			// code that is repeated every cycle in this state
				iCharacteristicAt2				:= aTransferPackages[0].iTransferValue;
				iCharacteristicAt4				:= aTransferPackages[1].iTransferValue;
				iOptProportionalGainFor2		:= aTransferPackages[2].iTransferValue;
				iOptIntegralGainFor2			:= aTransferPackages[3].iTransferValue;
				iOptTimeConstantFor2			:= aTransferPackages[4].iTransferValue;
				iOptShiftZeroPointSwitchOff2	:= aTransferPackages[5].iTransferValue;
				iOptProportionalGainFor4		:= aTransferPackages[6].iTransferValue;
				iOptIntegralGainFor4			:= aTransferPackages[7].iTransferValue;
				iOptTimeConstantFor4			:= aTransferPackages[8].iTransferValue;
				iOptShiftZeroPointSwitchOff4	:= aTransferPackages[9].iTransferValue;
				iInPortRetracted_optional		:= aTransferPackages[10].iTransferValue;
				iInPortAdvanced_optional		:= aTransferPackages[11].iTransferValue;
			//-----------------------------------------------------------------------------------------------------------
			
			// Transition
				xStateChange := TRUE;
				iState := 50;
				iCommandNumber := 40;
			//-----------------------------------------------------------------------------------------------------------
		
		50:	// DONE
			// code that is executed only in the first cycle of this state
				IF xStateChange = TRUE THEN
					xStateChange := FALSE;
					iResponse := eTransferResponse.transfer_successful;
					xDone := TRUE;
					xError := FALSE;
					xBusy := FALSE;
					xAborted := FALSE;
				END_IF
			//-----------------------------------------------------------------------------------------------------------
			
			// code that is repeated every cycle in this state	
				IF fbuploadMultipleParameters.xExecute = FALSE  AND fbuploadMultipleParameters.xUploadDone = FALSE AND fbuploadMultipleParameters.xUploadError = FALSE AND iCurrentValveMode = 63 THEN		//FB_UploadMultipleParameters was reset
					iCommandNumber := 5;	// exit transfer mode
				END_IF
			//-----------------------------------------------------------------------------------------------------------
			
			// Transition
				IF fbuploadMultipleParameters.xExecute = FALSE  AND fbuploadMultipleParameters.xUploadDone = FALSE AND fbuploadMultipleParameters.xUploadError = FALSE AND xExecute = FALSE THEN
					xStateChange := TRUE;
					iState := 100;
				END_IF
			//-----------------------------------------------------------------------------------------------------------
			
		70:	// ERROR
			// code that is executed only in the first cycle of this state
				IF xStateChange = TRUE THEN
					xStateChange := FALSE;
					//iResponse := eTransferResponse.communication_failed;	// set within the transition of the last state
					xDone := FALSE;
					xError := TRUE;
					xBusy := FALSE;
					xAborted := FALSE;
				END_IF
			//-----------------------------------------------------------------------------------------------------------
			
			// code that is repeated every cycle in this state	
			//-----------------------------------------------------------------------------------------------------------
			
			// Transition
				IF xExecute = FALSE AND xAbort = FALSE THEN
					xStateChange := TRUE;
					iState := 100;
				END_IF
			//-----------------------------------------------------------------------------------------------------------
			
		80:	// ABORTING
			// code that is executed only in the first cycle of this state
				IF xStateChange = TRUE THEN
					xStateChange := FALSE;
					iResponse := eTransferResponse.aborting;
					xBusy := FALSE;
					xDone := FALSE;
					xError := FALSE;
					xAborted := TRUE;
				END_IF
			//-----------------------------------------------------------------------------------------------------------
			
			// code that is repeated every cycle in this state
				IF iCurrentValveMode = 63 THEN
					iCommandNumber := 5;	// exit transfer mode
				ELSIF iCurrentValveMode <> 61 AND iCurrentValveMode <> 63 THEN
					iCommandNumber := 6;	// stop running motion apps
				ELSE
					iCommandNumber := 0; 
				END_IF
			//-----------------------------------------------------------------------------------------------------------
			
			// Transition
				IF xAbort = FALSE AND xExecute = FALSE AND iCurrentValveMode = 61 THEN
					xStateChange := TRUE;
					iState := 100;
				END_IF
			//-----------------------------------------------------------------------------------------------------------

		100:	// RESETTING FUNCTION BLOCK AND VALVE
			// code that is executed only in the first cycle of this state
				IF xStateChange = TRUE THEN
					xStateChange := FALSE;
					iResponse := eTransferResponse.resetting;
					xDone := FALSE;
					xError := FALSE;
					xBusy := FALSE;
					xAborted := FALSE;
				END_IF
			//-----------------------------------------------------------------------------------------------------------
			
			// code that is repeated every cycle in this state	
				IF iCurrentValveMode = 63 THEN
					iCommandNumber := 5;	// exit transfer mode
				ELSIF iCurrentValveMode <> 61 AND iCurrentValveMode <> 63 THEN
					iCommandNumber := 6;	// stop running motion apps
				END_IF
				
				// reset funktion block fbreadmultipleparameters
				// not done via command number because this is used to reset valve
					fbuploadMultipleParameters(
						awBusDataFromVTEM:= awBusDataFromVTEM, 
						awBusDataToVTEM:= awBusDataToVTEM, 
						xExecute:= FALSE, 
						iResponse=> , 
						iCurrentValue=> , 
						xUploadDone=> , 
						xUploadError=> , 
						aTransferPackages:= aTransferPackages);
				
				// reset parameter outputs
					iParameterSet := 1;
					iCharacteristicAt2 := 0;
					iCharacteristicAt4 := 0;
					iOptProportionalGainFor2 := 0;
					iOptIntegralGainFor2 := 0;
					iOptTimeConstantFor2 := 0;
					iOptShiftZeroPointSwitchOff2 := 0;
					iOptProportionalGainFor4 := 0;
					iOptIntegralGainFor4 := 0;
					iOptTimeConstantFor4 := 0;
					iOptShiftZeroPointSwitchOff4 := 0;
					iInPortRetracted_optional := 0;
					iInPortAdvanced_optional := 0;
				
				// reset parameter array
					FOR iCounterResetArray := 0 TO 100 BY 1 DO
						aTransferPackages[iCounterResetArray].iChannel := 0;
						aTransferPackages[iCounterResetArray].iAddressedTarget := 0;
						aTransferPackages[iCounterResetArray].iIndex := 0;
						aTransferPackages[iCounterResetArray].iTransferValue := 0;
					END_FOR
					
					iCounterResetArray := 0;
					xFirstCycle := TRUE;
			//-----------------------------------------------------------------------------------------------------------
			
			// Transition
				IF iCurrentValveMode = 61 THEN
					iCommandNumber := 6; // Last command to send before the FB is in IDLE
					xStateChange := TRUE;
					iState := 10;
				END_IF
			//-----------------------------------------------------------------------------------------------------------
			
	END_CASE
//-----------------------------------------------------------------------------------------------------------

// Command section
	CASE iCommandNumber OF
		0:	// IDLE
			;
		
		5:	// EXIT TRANSFER MODE
			fbwritevaluetoword(iValue:=63, iStartBit:=0, iEndBit:=5, wDataWord:=awBusDataToVTEM[0], xError=> );							// Valve Mode = 63
			fbwritevaluetoword(iValue:=0, iStartBit:=6, iEndBit:=7, wDataWord:=awBusDataToVTEM[0], xError=> );							// 0 (unused)
			fbwritevaluetoword(iValue:=0, iStartBit:=8, iEndBit:=12, wDataWord:=awBusDataToVTEM[0], xError=> );							// Channel = 0 (ignored)
			fbwritevaluetoword(iValue:=3, iStartBit:=13, iEndBit:=15, wDataWord:=awBusDataToVTEM[0], xError=> );						// Transfer Control = 3 (Exit transfer mode)
			fbwritevaluetoword(iValue:=0, iStartBit:=0, iEndBit:=7, wDataWord:=awBusDataToVTEM[1], xError=> );							// Addressed Target = 0 (ignored)
			fbwritevaluetoword(iValue:=0, iStartBit:=8, iEndBit:=15, wDataWord:=awBusDataToVTEM[1], xError=> );							// Index = 0 (ignored)
			fbwritevaluetoword(iValue:=0, iStartBit:=0, iEndBit:=15, wDataWord:=awBusDataToVTEM[2], xError=> );							// Value = 0 (ignored)
			
		6:	// STOP RUNNING MOTION APP
			fbwritevaluetoword(iValue:=61, iStartBit:=0, iEndBit:=5, wDataWord:=awBusDataToVTEM[0], xError=> );							// Valve Mode = 61 (stop)
			fbwritevaluetoword(iValue:=0, iStartBit:=6, iEndBit:=7, wDataWord:=awBusDataToVTEM[0], xError=> );							// App Control = 0 (unused)
			fbwritevaluetoword(iValue:=0, iStartBit:=8, iEndBit:=15, wDataWord:=awBusDataToVTEM[0], xError=> );							// App Option = 0 (unused)
			fbwritevaluetoword(iValue:=0, iStartBit:=0, iEndBit:=15, wDataWord:=awBusDataToVTEM[1], xError=> );							// Setpoint Value 1 = 0 (unused)
			fbwritevaluetoword(iValue:=0, iStartBit:=0, iEndBit:=15, wDataWord:=awBusDataToVTEM[2], xError=> );							// Setpoint Value 2 = 0 (unused)
		
		30:	// RUN FB_UPLOADMULTIPLEPARAMETERS
			fbuploadMultipleParameters(
				awBusDataFromVTEM:= awBusDataFromVTEM, 
				awBusDataToVTEM:= awBusDataToVTEM, 
				xExecute:= TRUE, 
				iResponse=> , 
				iCurrentValue=> , 
				xUploadDone=> , 
				xUploadError=> , 
				aTransferPackages:= aTransferPackages);

		40:	// RESET FB_UPLOADMULTIPLEPARAMETERS
			fbuploadMultipleParameters(
				awBusDataFromVTEM:= awBusDataFromVTEM, 
				awBusDataToVTEM:= awBusDataToVTEM, 
				xExecute:= FALSE, 
				iResponse=> , 
				iCurrentValue=> , 
				xUploadDone=> , 
				xUploadError=> , 
				aTransferPackages:= aTransferPackages);
	END_CASE
//-----------------------------------------------------------------------------------------------------------

END_FUNCTION_BLOCK

// Transfermode/specific_MA_config/FB_Read_config_MA_04
/// This function block can be used to upload the configuration of Motion App 4 ("Model-based proportional pressure regulation").
/// The specific parameters of this Motion App are the outputs of this FB
/// The function block uses the transfer mode to read this configuration from the Motion Terminal
/// and indicates the state of the upload process at the output iResponse.

FUNCTION_BLOCK FB_Read_config_MA_04
VAR_INPUT
	awBusDataFromVTEM 				: ARRAY [0..2] OF WORD;		// array of 3 words of process data received from the Motion Terminal
END_VAR
	
VAR_IN_OUT
	awBusDataToVTEM 				: ARRAY [0..2] OF WORD; 	// array of 3 words of process data sent to the Motion Terminal
END_VAR

VAR_INPUT
	xExecute 						: BOOL; 					// rising edge starts the reading process, falling edge resets the function block after reading is done
	xAbort							: BOOL;						// rising edge aborts the reading process
	iParameterSet					: INT := 1; 				// the parameter set to be read from, 1 by default
END_VAR                     		

VAR_OUTPUT                  		
	// system parameters
		iTubingLengthAt2 			: INT; 						// length of the tubing connected to outlet port 2 of the valve [1 digit = 1 mm]
		iTubingLengthAt4 			: INT;						// length of the tubing connected to outlet port 4 of the valve [1 digit = 1 mm]
		iTubingInnerDiameterAt2 	: INT;  					// inner diameter of the tubing connected to outlet port 2 of the valve [1 digit = 0.01 mm]
		iTubingInnerDiameterAt4 	: INT;						// inner diameter of the tubing connected to outlet port 4 of the valve [1 digit = 0.01 mm]
		iVolumeAt2 					: INT; 						// size/capacity of the volume connected to outlet port 2 of the valve [1 digit = 0.001 l]
	 	iVolumeAt4 					: INT;						// size/capacity of the volume connected to outlet port 4 of the valve [1 digit = 0.001 l]
		iInPortRetracted_optional	: INT;						// Sensor port for detection of end position at pressurisation of outlet port 2 (retracted), value is number of the slot (beginning from 0 and including valve slots) * 10 + number of the port
		iInPortAdvanced_optional	: INT;						// Sensor port for detection of end position at pressurisation of outlet port 4 (advanced), value is number of the slot (beginning from 0 and including valve slots) * 10 + number of the port
		
	// application parameters
		iPressureRiseAt2 			: INT; 						// maximum pressure rise at outlet port 2 [1 digit = 0.01 bar/s]
		iPressureRiseAt4 			: INT;						// maximum pressure rise at outlet port 4 [1 digit = 0.01 bar/s]
		
	// function block response
		iResponse 					: eTransferResponse; 		// returns the status of the upload process
		xBusy						: BOOL;						// TRUE as long as the upload process is running
		xDone 						: BOOL; 					// indicates whether the upload was successfull
		xError 						: BOOL; 					// indicates whether an error occurred during the transfer
		xAborted					: BOOL;						// TRUE if the function block was canceled by xAbort	
END_VAR

VAR
	iState							: INT := 10;
	xStateChange					: BOOL;
	iCommandNumber					: INT;
	xFirstCycle						: BOOL := TRUE;				// indicator for the first cycle of the function block
	iParameterSetFC					: INT;						// value on input iParameterSet during first cycle
	
	aTransferPackages				: ARRAY [0..100] OF stTransferPackage;
	fbreadbitsfromword				: FB_Read_Bits_From_Word;
	fbuploadMultipleParameters 		: FB_Upload_Multiple_Parameters;
	fbWriteValueToWord 				: FB_Write_Value_To_Word;

	iCounterResetArray				: INT;

	iCurrentValveMode				: INT;						//
END_VAR

(*****************************************************************************************************

Festo SE & Co. KG, Esslingen
Copyright (c) 2021. All rights reserved.

Product:            Motion Terminal VTEM
Description:        Function Block to upload the parameters for Motion App 4 from the Motion Terminal

Object version:     2.00
Last change:        2021-07
======================================================================================================
                                       H I S T O R Y
======================================================================================================
Version:            2.00
Date:               2021-07
Change/Activity:    - created (#3872357)
Release:            3.5.7.237 (CODESYS 3.5.7.2, Lib version 3.7)
Author:             JEBU
======================================================================================================

*****************************************************************************************************)

// pre-check of the value for the parameter set
	IF xExecute = TRUE AND (iParameterSet < 1 OR iParameterSet > 5) THEN		// invalid input for the parameter set
		xDone := FALSE; 
		xError := TRUE; 
		iResponse := eTransferResponse.invalid_ParameterSet;
		xStateChange := TRUE;
		iState := 70;	// ERROR
	END_IF
//-----------------------------------------------------------------------------------------------------------

// check if iParameterSet was changed
	IF xExecute = TRUE AND xFirstCycle = TRUE THEN
		xFirstCycle := FALSE;
		iParameterSetFC := iParameterSet;
	END_IF
	
	IF xExecute = TRUE AND iParameterSet <> iParameterSetFC THEN
		xStateChange := TRUE;
		iState := 70;
		iResponse := eTransferResponse.FB_needs_rising_edge_xExecute;
	END_IF
//-----------------------------------------------------------------------------------------------------------

// WRITE PARAMETER INDICES INTO ARRAY
	//iTubingLengthAt2
		aTransferPackages[0].iChannel := iParameterSet;
		aTransferPackages[0].iAddressedTarget := 4;
		aTransferPackages[0].iIndex := 12;
	
	//iTubingLengthAt4
		aTransferPackages[1].iChannel := iParameterSet;
		aTransferPackages[1].iAddressedTarget := 4;
		aTransferPackages[1].iIndex := 13;
	
	//iTubingInnerDiameterAt2
		aTransferPackages[2].iChannel := iParameterSet;
		aTransferPackages[2].iAddressedTarget := 4;
		aTransferPackages[2].iIndex := 14;
	
	//iTubingInnerDiameterAt4
		aTransferPackages[3].iChannel := iParameterSet;
		aTransferPackages[3].iAddressedTarget := 4;
		aTransferPackages[3].iIndex := 15;
	
	//iVolumeAt2
		aTransferPackages[4].iChannel := iParameterSet;
		aTransferPackages[4].iAddressedTarget := 4;
		aTransferPackages[4].iIndex := 40;
	
	//iVolumeAt4
		aTransferPackages[5].iChannel := iParameterSet;
		aTransferPackages[5].iAddressedTarget := 4;
		aTransferPackages[5].iIndex := 41;
	
	//iPressureRiseAt2
		aTransferPackages[6].iChannel := iParameterSet;
		aTransferPackages[6].iAddressedTarget := 4;
		aTransferPackages[6].iIndex := 182;
	
	//iPressureRiseAt4
		aTransferPackages[7].iChannel := iParameterSet;
		aTransferPackages[7].iAddressedTarget := 4;
		aTransferPackages[7].iIndex := 183;
	
	//iInPortRetract_optional
		aTransferPackages[8].iChannel := iParameterSet;
		aTransferPackages[8].iAddressedTarget := 4;
		aTransferPackages[8].iIndex := 70;
	
	//iInPortAdvanced_optional
		aTransferPackages[9].iChannel := iParameterSet;
		aTransferPackages[9].iAddressedTarget := 4;
		aTransferPackages[9].iIndex := 71;
	
	// define end of parameter list to be uploaded by setting all variables to 0 (end criterion for FB_Upload_Multiple_Parameters)
		aTransferPackages[10].iChannel := 0;
		aTransferPackages[10].iAddressedTarget := 0;
		aTransferPackages[10].iIndex := 0;
//-----------------------------------------------------------------------------------------------------------

// Read the current status of the the motion terminal
	fbreadbitsfromword(wData:= awBusDataFromVTEM[0], iStartBit:=0, iEndBit:= 5, iValue=> iCurrentValveMode, xError=> );				// read current valve mode
//-----------------------------------------------------------------------------------------------------------

// Transition: Aborting condition when xAbort is TRUE in all States except "IDLE" , "ABORTING" and "RESETTING"
	IF xAbort = TRUE AND NOT(iState = 10 AND xExecute = FALSE) AND iState <> 80 AND iState <> 100 THEN
		xStateChange := TRUE;	// Leaving current state
		iState := 80;	// Choosing next state, here: ABORTING
	END_IF
//-----------------------------------------------------------------------------------------------------------

// local state machine
	CASE iState OF
		10:	// IDLE
			// code that is executed only in the first cycle of this state
				IF xStateChange = TRUE THEN
					xStateChange := FALSE;
					iResponse := eTransferResponse.ready_for_new_transfer;
					xDone := FALSE;
					xError := FALSE;
					xBusy := FALSE;
					xAborted := FALSE;
				END_IF
			//-----------------------------------------------------------------------------------------------------------
			
			// code that is repeated every cycle in this state
				iCommandNumber := 0;
			//-----------------------------------------------------------------------------------------------------------
			
			// Transition
			IF xExecute = TRUE THEN
				xStateChange := TRUE;
				iState := 20;
			END_IF
			//-----------------------------------------------------------------------------------------------------------
		
		20:	// RESETTING VALVE MODE TO 61
			// code that is executed only in the first cycle of this state
				IF xStateChange = TRUE THEN
					xStateChange := FALSE;
					iResponse := eTransferResponse.preparing_transfer;
					xDone := FALSE;
					xError := FALSE;
					xBusy := TRUE;
					xAborted := FALSE;
				END_IF
			//-----------------------------------------------------------------------------------------------------------
			
			// code that is repeated every cycle in this state	
				IF iCurrentValveMode = 63 THEN
					iCommandNumber := 5;	// exit transfer mode
				ELSIF iCurrentValveMode <> 61 AND iCurrentValveMode <> 63 THEN
					iCommandNumber := 6;	// stop running motion apps
				END_IF 
			//-----------------------------------------------------------------------------------------------------------
			
			// Transition
				IF iCurrentValveMode = 61 THEN
					xStateChange := TRUE;	// Leave this state
					iState := 30;
					iCommandNumber := 30;			
				END_IF
			//-----------------------------------------------------------------------------------------------------------
		
		30:	// READING PARAMETER VALUES
			// code that is executed only in the first cycle of this state
				IF xStateChange = TRUE THEN
					xStateChange := FALSE;
					iResponse := eTransferResponse.transferring;
					xDone := FALSE;
					xError := FALSE;
					xBusy := TRUE;
					xAborted := FALSE;
				END_IF
			//-----------------------------------------------------------------------------------------------------------
			
			// code that is repeated every cycle in this state
				iCommandNumber := 30;		// read parameter values
			//-----------------------------------------------------------------------------------------------------------
			
			// Transition
				IF fbuploadMultipleParameters.xExecute = TRUE AND fbuploadMultipleParameters.xUploadDone = TRUE AND fbuploadMultipleParameters.xUploadError = FALSE THEN	// Upload Done
					xStateChange := TRUE;
					iState := 40;	// Write parameter values to outputs
				ELSIF fbuploadMultipleParameters.xExecute = TRUE AND fbuploadMultipleParameters.xUploadDone = FALSE AND fbuploadMultipleParameters.xUploadError = TRUE THEN	// Error during update
					xStateChange := TRUE;
					iState := 70;	// ERROR
					iResponse := fbuploadMultipleParameters.iResponse;
				END_IF
			//-----------------------------------------------------------------------------------------------------------
		
		40:	// WRITE PARAMETER VALUES TO OUTPUTS
			// code that is executed only in the first cycle of this state
				IF xStateChange = TRUE THEN
					xStateChange := FALSE;
					iResponse := eTransferResponse.transferring;
					xDone := FALSE;
					xError := FALSE;
					xBusy := TRUE;
					xAborted := FALSE;
				END_IF
			//-----------------------------------------------------------------------------------------------------------
			
			// code that is repeated every cycle in this state
				iTubingLengthAt2			:= aTransferPackages[0].iTransferValue;
				iTubingLengthAt4			:= aTransferPackages[1].iTransferValue;
				iTubingInnerDiameterAt2		:= aTransferPackages[2].iTransferValue;
				iTubingInnerDiameterAt4		:= aTransferPackages[3].iTransferValue;
				iVolumeAt2					:= aTransferPackages[4].iTransferValue;
				iVolumeAt4					:= aTransferPackages[5].iTransferValue;
				iPressureRiseAt2			:= aTransferPackages[6].iTransferValue;
				iPressureRiseAt4			:= aTransferPackages[7].iTransferValue;
				iInPortRetracted_optional	:= aTransferPackages[8].iTransferValue;
				iInPortAdvanced_optional	:= aTransferPackages[9].iTransferValue;
			//-----------------------------------------------------------------------------------------------------------
			
			// Transition
				xStateChange := TRUE;
				iState := 50;
				iCommandNumber := 40;
			//-----------------------------------------------------------------------------------------------------------
		
		50:	// DONE
			// code that is executed only in the first cycle of this state
				IF xStateChange = TRUE THEN
					xStateChange := FALSE;
					iResponse := eTransferResponse.transfer_successful;
					xDone := TRUE;
					xError := FALSE;
					xBusy := FALSE;
					xAborted := FALSE;
				END_IF
			//-----------------------------------------------------------------------------------------------------------
			
			// code that is repeated every cycle in this state	
				IF fbuploadMultipleParameters.xExecute = FALSE  AND fbuploadMultipleParameters.xUploadDone = FALSE AND fbuploadMultipleParameters.xUploadError = FALSE AND iCurrentValveMode = 63 THEN		//FB_UploadMultipleParameters was reset
					iCommandNumber := 5;	// exit transfer mode
				END_IF
			//-----------------------------------------------------------------------------------------------------------
			
			// Transition
				IF fbuploadMultipleParameters.xExecute = FALSE  AND fbuploadMultipleParameters.xUploadDone = FALSE AND fbuploadMultipleParameters.xUploadError = FALSE AND xExecute = FALSE THEN
					xStateChange := TRUE;
					iState := 100;
				END_IF
			//-----------------------------------------------------------------------------------------------------------
			
		70:	// ERROR
			// code that is executed only in the first cycle of this state
				IF xStateChange = TRUE THEN
					xStateChange := FALSE;
					//iResponse := eTransferResponse.communication_failed;	// set within the transition of the last state
					xDone := FALSE;
					xError := TRUE;
					xBusy := FALSE;
					xAborted := FALSE;
				END_IF
			//-----------------------------------------------------------------------------------------------------------
			
			// code that is repeated every cycle in this state	
			//-----------------------------------------------------------------------------------------------------------
			
			// Transition
				IF xExecute = FALSE AND xAbort = FALSE THEN
					xStateChange := TRUE;
					iState := 100;
				END_IF
			//-----------------------------------------------------------------------------------------------------------
			
		80:	// ABORTING
			// code that is executed only in the first cycle of this state
				IF xStateChange = TRUE THEN
					xStateChange := FALSE;
					iResponse := eTransferResponse.aborting;
					xBusy := FALSE;
					xDone := FALSE;
					xError := FALSE;
					xAborted := TRUE;
				END_IF
			//-----------------------------------------------------------------------------------------------------------
			
			// code that is repeated every cycle in this state
				IF iCurrentValveMode = 63 THEN
					iCommandNumber := 5;	// exit transfer mode
				ELSIF iCurrentValveMode <> 61 AND iCurrentValveMode <> 63 THEN
					iCommandNumber := 6;	// stop running motion apps
				ELSE
					iCommandNumber := 0; 
				END_IF
			//-----------------------------------------------------------------------------------------------------------
			
			// Transition
				IF xAbort = FALSE AND xExecute = FALSE AND iCurrentValveMode = 61 THEN
					xStateChange := TRUE;
					iState := 100;
				END_IF
			//-----------------------------------------------------------------------------------------------------------

		100:	// RESETTING FUNCTION BLOCK AND VALVE
			// code that is executed only in the first cycle of this state
				IF xStateChange = TRUE THEN
					xStateChange := FALSE;
					iResponse := eTransferResponse.resetting;
					xDone := FALSE;
					xError := FALSE;
					xBusy := FALSE;
					xAborted := FALSE;
				END_IF
			//-----------------------------------------------------------------------------------------------------------
			
			// code that is repeated every cycle in this state	
				IF iCurrentValveMode = 63 THEN
					iCommandNumber := 5;	// exit transfer mode
				ELSIF iCurrentValveMode <> 61 AND iCurrentValveMode <> 63 THEN
					iCommandNumber := 6;	// stop running motion apps
				END_IF
				
				// reset funktion block fbreadmultipleparameters
				// not done via command number because this is used to reset valve
					fbuploadMultipleParameters(
						awBusDataFromVTEM:= awBusDataFromVTEM, 
						awBusDataToVTEM:= awBusDataToVTEM, 
						xExecute:= FALSE, 
						iResponse=> , 
						iCurrentValue=> , 
						xUploadDone=> , 
						xUploadError=> , 
						aTransferPackages:= aTransferPackages);
				
				// reset parameter outputs
					iParameterSet				:= 1;
					iTubingLengthAt2			:= 0;
					iTubingLengthAt4			:= 0;
					iTubingInnerDiameterAt2		:= 0;
					iTubingInnerDiameterAt4		:= 0;
					iVolumeAt2					:= 0;
					iVolumeAt4					:= 0;
					iPressureRiseAt2			:= 0;
					iPressureRiseAt4			:= 0;
					iInPortRetracted_optional	:= 0;
					iInPortAdvanced_optional	:= 0;
				
				// reset parameter array
					FOR iCounterResetArray := 0 TO 100 BY 1 DO
						aTransferPackages[iCounterResetArray].iChannel := 0;
						aTransferPackages[iCounterResetArray].iAddressedTarget := 0;
						aTransferPackages[iCounterResetArray].iIndex := 0;
						aTransferPackages[iCounterResetArray].iTransferValue := 0;
					END_FOR
					
					iCounterResetArray := 0;
					xFirstCycle := TRUE;
			//-----------------------------------------------------------------------------------------------------------
			
			// Transition
				IF iCurrentValveMode = 61 THEN
					iCommandNumber := 6; // Last command to send before the FB is in IDLE
					xStateChange := TRUE;
					iState := 10;
				END_IF
			//-----------------------------------------------------------------------------------------------------------
			
	END_CASE
//-----------------------------------------------------------------------------------------------------------

// Command section
	CASE iCommandNumber OF
		0:	// IDLE
			;
		
		5:	// EXIT TRANSFER MODE
			fbwritevaluetoword(iValue:=63, iStartBit:=0, iEndBit:=5, wDataWord:=awBusDataToVTEM[0], xError=> );							// Valve Mode = 63
			fbwritevaluetoword(iValue:=0, iStartBit:=6, iEndBit:=7, wDataWord:=awBusDataToVTEM[0], xError=> );							// 0 (unused)
			fbwritevaluetoword(iValue:=0, iStartBit:=8, iEndBit:=12, wDataWord:=awBusDataToVTEM[0], xError=> );							// Channel = 0 (ignored)
			fbwritevaluetoword(iValue:=3, iStartBit:=13, iEndBit:=15, wDataWord:=awBusDataToVTEM[0], xError=> );						// Transfer Control = 3 (Exit transfer mode)
			fbwritevaluetoword(iValue:=0, iStartBit:=0, iEndBit:=7, wDataWord:=awBusDataToVTEM[1], xError=> );							// Addressed Target = 0 (ignored)
			fbwritevaluetoword(iValue:=0, iStartBit:=8, iEndBit:=15, wDataWord:=awBusDataToVTEM[1], xError=> );							// Index = 0 (ignored)
			fbwritevaluetoword(iValue:=0, iStartBit:=0, iEndBit:=15, wDataWord:=awBusDataToVTEM[2], xError=> );							// Value = 0 (ignored)
			
		6:	// STOP RUNNING MOTION APP
			fbwritevaluetoword(iValue:=61, iStartBit:=0, iEndBit:=5, wDataWord:=awBusDataToVTEM[0], xError=> );							// Valve Mode = 61 (stop)
			fbwritevaluetoword(iValue:=0, iStartBit:=6, iEndBit:=7, wDataWord:=awBusDataToVTEM[0], xError=> );							// App Control = 0 (unused)
			fbwritevaluetoword(iValue:=0, iStartBit:=8, iEndBit:=15, wDataWord:=awBusDataToVTEM[0], xError=> );							// App Option = 0 (unused)
			fbwritevaluetoword(iValue:=0, iStartBit:=0, iEndBit:=15, wDataWord:=awBusDataToVTEM[1], xError=> );							// Setpoint Value 1 = 0 (unused)
			fbwritevaluetoword(iValue:=0, iStartBit:=0, iEndBit:=15, wDataWord:=awBusDataToVTEM[2], xError=> );							// Setpoint Value 2 = 0 (unused)
		
		30:	// RUN FB_UPLOADMULTIPLEPARAMETERS
			fbuploadMultipleParameters(
				awBusDataFromVTEM:= awBusDataFromVTEM, 
				awBusDataToVTEM:= awBusDataToVTEM, 
				xExecute:= TRUE, 
				iResponse=> , 
				iCurrentValue=> , 
				xUploadDone=> , 
				xUploadError=> , 
				aTransferPackages:= aTransferPackages);

		40:	// RESET FB_UPLOADMULTIPLEPARAMETERS
			fbuploadMultipleParameters(
				awBusDataFromVTEM:= awBusDataFromVTEM, 
				awBusDataToVTEM:= awBusDataToVTEM, 
				xExecute:= FALSE, 
				iResponse=> , 
				iCurrentValue=> , 
				xUploadDone=> , 
				xUploadError=> , 
				aTransferPackages:= aTransferPackages);
	END_CASE
//-----------------------------------------------------------------------------------------------------------

END_FUNCTION_BLOCK

// Transfermode/specific_MA_config/FB_Read_config_MA_05
/// This function block can be used to upload the configuration of Motion App 5 ("Supply and exhaust air flow control").
/// The specific parameters of this Motion App are the outputs of this FB
/// The function block uses the transfer mode to read this configuration from the Motion Terminal
/// and indicates the state of the upload process at the output iResponse.

FUNCTION_BLOCK FB_Read_config_MA_05
VAR_INPUT
	awBusDataFromVTEM 				: ARRAY [0..2] OF WORD;		// array of 3 words of process data received from the Motion Terminal
END_VAR
	
VAR_IN_OUT
	awBusDataToVTEM 				: ARRAY [0..2] OF WORD; 	// array of 3 words of process data sent to the Motion Terminal
END_VAR

VAR_INPUT
	xExecute 						: BOOL; 					// rising edge starts the reading process, falling edge resets the function block after reading is done
	xAbort							: BOOL;						// rising edge aborts the reading process
	iParameterSet					: INT := 1; 				// the parameter set to be read from, 1 by default
END_VAR                     		

VAR_OUTPUT                  		
	// system parameters
		iInPortRetracted_optional	: INT;						// Sensor port for detection of end position at pressurisation of outlet port 2 (retracted), value is number of the slot (beginning from 0 and including valve slots) * 10 + number of the port
		iInPortAdvanced_optional	: INT;						// Sensor port for detection of end position at pressurisation of outlet port 4 (advanced), value is number of the slot (beginning from 0 and including valve slots) * 10 + number of the port

	// application parameters                       	
		iSoftStartFunction			: INT;						// flag to enable or disable the SoftStartFunction; 0 = disabled, 1 = enabled
		
	// function block response
		iResponse 					: eTransferResponse; 		// returns the status of the upload process
		xBusy						: BOOL;						// TRUE as long as the upload process is running
		xDone 						: BOOL; 					// indicates whether the upload was successfull
		xError 						: BOOL; 					// indicates whether an error occurred during the transfer
		xAborted					: BOOL;						// TRUE if the function block was canceled by xAbort	
END_VAR

VAR
	iState							: INT := 10;
	xStateChange					: BOOL;
	iCommandNumber					: INT;
	xFirstCycle						: BOOL := TRUE;				// indicator for the first cycle of the function block
	iParameterSetFC					: INT;						// value on input iParameterSet during first cycle
	
	aTransferPackages				: ARRAY [0..100] OF stTransferPackage;
	fbreadbitsfromword				: FB_Read_Bits_From_Word;
	fbuploadMultipleParameters 		: FB_Upload_Multiple_Parameters;
	fbWriteValueToWord 				: FB_Write_Value_To_Word;

	iCounterResetArray				: INT;

	iCurrentValveMode				: INT;						//
END_VAR

(*****************************************************************************************************

Festo SE & Co. KG, Esslingen
Copyright (c) 2021. All rights reserved.

Product:            Motion Terminal VTEM
Description:        Function Block to upload the parameters for Motion App 5 from the Motion Terminal

Object version:     2.00
Last change:        2021-07
======================================================================================================
                                       H I S T O R Y
======================================================================================================
Version:            2.00
Date:               2021-07
Change/Activity:    - created (#3872357)
Release:            3.5.7.237 (CODESYS 3.5.7.2, Lib version 3.7)
Author:             JEBU
======================================================================================================

*****************************************************************************************************)

// pre-check of the value for the parameter set
	IF xExecute = TRUE AND (iParameterSet < 1 OR iParameterSet > 5) THEN		// invalid input for the parameter set
		xDone := FALSE; 
		xError := TRUE; 
		iResponse := eTransferResponse.invalid_ParameterSet;
		xStateChange := TRUE;
		iState := 70;	// ERROR
	END_IF
//-----------------------------------------------------------------------------------------------------------

// check if iParameterSet was changed
	IF xExecute = TRUE AND xFirstCycle = TRUE THEN
		xFirstCycle := FALSE;
		iParameterSetFC := iParameterSet;
	END_IF
	
	IF xExecute = TRUE AND iParameterSet <> iParameterSetFC THEN
		xStateChange := TRUE;
		iState := 70;
		iResponse := eTransferResponse.FB_needs_rising_edge_xExecute;
	END_IF
//-----------------------------------------------------------------------------------------------------------

// WRITE PARAMETER INDICES INTO ARRAY
	//iSoftStartFunction
		aTransferPackages[0].iChannel := iParameterSet;
		aTransferPackages[0].iAddressedTarget := 5;
		aTransferPackages[0].iIndex := 222;
	
	//iInPortRetract_optional
		aTransferPackages[1].iChannel := iParameterSet;
		aTransferPackages[1].iAddressedTarget := 5;
		aTransferPackages[1].iIndex := 70;
	
	//iInPortAdvanced_optional
		aTransferPackages[2].iChannel := iParameterSet;
		aTransferPackages[2].iAddressedTarget := 5;
		aTransferPackages[2].iIndex := 71;
	
	// define end of parameter list to be uploaded by setting all variables to 0 (end criterion for FB_Upload_Multiple_Parameters)
		aTransferPackages[3].iChannel := 0;
		aTransferPackages[3].iAddressedTarget := 0;
		aTransferPackages[3].iIndex := 0;
//-----------------------------------------------------------------------------------------------------------

// Read the current status of the the motion terminal
	fbreadbitsfromword(wData:= awBusDataFromVTEM[0], iStartBit:=0, iEndBit:= 5, iValue=> iCurrentValveMode, xError=> );				// read current valve mode
//-----------------------------------------------------------------------------------------------------------

// Transition: Aborting condition when xAbort is TRUE in all States except "IDLE" , "ABORTING" and "RESETTING"
	IF xAbort = TRUE AND NOT(iState = 10 AND xExecute = FALSE) AND iState <> 80 AND iState <> 100 THEN
		xStateChange := TRUE;	// Leaving current state
		iState := 80;	// Choosing next state, here: ABORTING
	END_IF
//-----------------------------------------------------------------------------------------------------------

// local state machine
	CASE iState OF
		10:	// IDLE
			// code that is executed only in the first cycle of this state
				IF xStateChange = TRUE THEN
					xStateChange := FALSE;
					iResponse := eTransferResponse.ready_for_new_transfer;
					xDone := FALSE;
					xError := FALSE;
					xBusy := FALSE;
					xAborted := FALSE;
				END_IF
			//-----------------------------------------------------------------------------------------------------------
			
			// code that is repeated every cycle in this state
				iCommandNumber := 0;
			//-----------------------------------------------------------------------------------------------------------
			
			// Transition
			IF xExecute = TRUE THEN
				xStateChange := TRUE;
				iState := 20;
			END_IF
			//-----------------------------------------------------------------------------------------------------------
		
		20:	// RESETTING VALVE MODE TO 61
			// code that is executed only in the first cycle of this state
				IF xStateChange = TRUE THEN
					xStateChange := FALSE;
					iResponse := eTransferResponse.preparing_transfer;
					xDone := FALSE;
					xError := FALSE;
					xBusy := TRUE;
					xAborted := FALSE;
				END_IF
			//-----------------------------------------------------------------------------------------------------------
			
			// code that is repeated every cycle in this state	
				IF iCurrentValveMode = 63 THEN
					iCommandNumber := 5;	// exit transfer mode
				ELSIF iCurrentValveMode <> 61 AND iCurrentValveMode <> 63 THEN
					iCommandNumber := 6;	// stop running motion apps
				END_IF 
			//-----------------------------------------------------------------------------------------------------------
			
			// Transition
				IF iCurrentValveMode = 61 THEN
					xStateChange := TRUE;	// Leave this state
					iState := 30;
					iCommandNumber := 30;			
				END_IF
			//-----------------------------------------------------------------------------------------------------------
		
		30:	// READING PARAMETER VALUES
			// code that is executed only in the first cycle of this state
				IF xStateChange = TRUE THEN
					xStateChange := FALSE;
					iResponse := eTransferResponse.transferring;
					xDone := FALSE;
					xError := FALSE;
					xBusy := TRUE;
					xAborted := FALSE;
				END_IF
			//-----------------------------------------------------------------------------------------------------------
			
			// code that is repeated every cycle in this state
				iCommandNumber := 30;		// read parameter values
			//-----------------------------------------------------------------------------------------------------------
			
			// Transition
				IF fbuploadMultipleParameters.xExecute = TRUE AND fbuploadMultipleParameters.xUploadDone = TRUE AND fbuploadMultipleParameters.xUploadError = FALSE THEN	// Upload Done
					xStateChange := TRUE;
					iState := 40;	// Write parameter values to outputs
				ELSIF fbuploadMultipleParameters.xExecute = TRUE AND fbuploadMultipleParameters.xUploadDone = FALSE AND fbuploadMultipleParameters.xUploadError = TRUE THEN	// Error during update
					xStateChange := TRUE;
					iState := 70;	// ERROR
					iResponse := fbuploadMultipleParameters.iResponse;
				END_IF
			//-----------------------------------------------------------------------------------------------------------
		
		40:	// WRITE PARAMETER VALUES TO OUTPUTS
			// code that is executed only in the first cycle of this state
				IF xStateChange = TRUE THEN
					xStateChange := FALSE;
					iResponse := eTransferResponse.transferring;
					xDone := FALSE;
					xError := FALSE;
					xBusy := TRUE;
					xAborted := FALSE;
				END_IF
			//-----------------------------------------------------------------------------------------------------------
			
			// code that is repeated every cycle in this state
				iSoftStartFunction			:= aTransferPackages[0].iTransferValue;
				iInPortRetracted_optional	:= aTransferPackages[1].iTransferValue;
				iInPortAdvanced_optional	:= aTransferPackages[2].iTransferValue;
			//-----------------------------------------------------------------------------------------------------------
			
			// Transition
				xStateChange := TRUE;
				iState := 50;
				iCommandNumber := 40;
			//-----------------------------------------------------------------------------------------------------------
		
		50:	// DONE
			// code that is executed only in the first cycle of this state
				IF xStateChange = TRUE THEN
					xStateChange := FALSE;
					iResponse := eTransferResponse.transfer_successful;
					xDone := TRUE;
					xError := FALSE;
					xBusy := FALSE;
					xAborted := FALSE;
				END_IF
			//-----------------------------------------------------------------------------------------------------------
			
			// code that is repeated every cycle in this state	
				IF fbuploadMultipleParameters.xExecute = FALSE  AND fbuploadMultipleParameters.xUploadDone = FALSE AND fbuploadMultipleParameters.xUploadError = FALSE AND iCurrentValveMode = 63 THEN		//FB_UploadMultipleParameters was reset
					iCommandNumber := 5;	// exit transfer mode
				END_IF
			//-----------------------------------------------------------------------------------------------------------
			
			// Transition
				IF fbuploadMultipleParameters.xExecute = FALSE  AND fbuploadMultipleParameters.xUploadDone = FALSE AND fbuploadMultipleParameters.xUploadError = FALSE AND xExecute = FALSE THEN
					xStateChange := TRUE;
					iState := 100;
				END_IF
			//-----------------------------------------------------------------------------------------------------------
			
		70:	// ERROR
			// code that is executed only in the first cycle of this state
				IF xStateChange = TRUE THEN
					xStateChange := FALSE;
					//iResponse := eTransferResponse.communication_failed;	// set within the transition of the last state
					xDone := FALSE;
					xError := TRUE;
					xBusy := FALSE;
					xAborted := FALSE;
				END_IF
			//-----------------------------------------------------------------------------------------------------------
			
			// code that is repeated every cycle in this state	
			//-----------------------------------------------------------------------------------------------------------
			
			// Transition
				IF xExecute = FALSE AND xAbort = FALSE THEN
					xStateChange := TRUE;
					iState := 100;
				END_IF
			//-----------------------------------------------------------------------------------------------------------
			
		80:	// ABORTING
			// code that is executed only in the first cycle of this state
				IF xStateChange = TRUE THEN
					xStateChange := FALSE;
					iResponse := eTransferResponse.aborting;
					xBusy := FALSE;
					xDone := FALSE;
					xError := FALSE;
					xAborted := TRUE;
				END_IF
			//-----------------------------------------------------------------------------------------------------------
			
			// code that is repeated every cycle in this state
				IF iCurrentValveMode = 63 THEN
					iCommandNumber := 5;	// exit transfer mode
				ELSIF iCurrentValveMode <> 61 AND iCurrentValveMode <> 63 THEN
					iCommandNumber := 6;	// stop running motion apps
				ELSE
					iCommandNumber := 0; 
				END_IF
			//-----------------------------------------------------------------------------------------------------------
			
			// Transition
				IF xAbort = FALSE AND xExecute = FALSE AND iCurrentValveMode = 61 THEN
					xStateChange := TRUE;
					iState := 100;
				END_IF
			//-----------------------------------------------------------------------------------------------------------

		100:	// RESETTING FUNCTION BLOCK AND VALVE
			// code that is executed only in the first cycle of this state
				IF xStateChange = TRUE THEN
					xStateChange := FALSE;
					iResponse := eTransferResponse.resetting;
					xDone := FALSE;
					xError := FALSE;
					xBusy := FALSE;
					xAborted := FALSE;
				END_IF
			//-----------------------------------------------------------------------------------------------------------
			
			// code that is repeated every cycle in this state	
				IF iCurrentValveMode = 63 THEN
					iCommandNumber := 5;	// exit transfer mode
				ELSIF iCurrentValveMode <> 61 AND iCurrentValveMode <> 63 THEN
					iCommandNumber := 6;	// stop running motion apps
				END_IF
				
				// reset funktion block fbreadmultipleparameters
				// not done via command number because this is used to reset valve
					fbuploadMultipleParameters(
						awBusDataFromVTEM:= awBusDataFromVTEM, 
						awBusDataToVTEM:= awBusDataToVTEM, 
						xExecute:= FALSE, 
						iResponse=> , 
						iCurrentValue=> , 
						xUploadDone=> , 
						xUploadError=> , 
						aTransferPackages:= aTransferPackages);
				
				// reset parameter outputs
					iParameterSet				:= 1;

					iSoftStartFunction			:= 0;
					iInPortRetracted_optional	:= 0;
					iInPortAdvanced_optional	:= 0;
				
				// reset parameter array
					FOR iCounterResetArray := 0 TO 100 BY 1 DO
						aTransferPackages[iCounterResetArray].iChannel := 0;
						aTransferPackages[iCounterResetArray].iAddressedTarget := 0;
						aTransferPackages[iCounterResetArray].iIndex := 0;
						aTransferPackages[iCounterResetArray].iTransferValue := 0;
					END_FOR
					
					iCounterResetArray := 0;
					xFirstCycle := TRUE;
			//-----------------------------------------------------------------------------------------------------------
			
			// Transition
				IF iCurrentValveMode = 61 THEN
					iCommandNumber := 6; // Last command to send before the FB is in IDLE
					xStateChange := TRUE;
					iState := 10;
				END_IF
			//-----------------------------------------------------------------------------------------------------------
			
	END_CASE
//-----------------------------------------------------------------------------------------------------------

// Command section
	CASE iCommandNumber OF
		0:	// IDLE
			;
		
		5:	// EXIT TRANSFER MODE
			fbwritevaluetoword(iValue:=63, iStartBit:=0, iEndBit:=5, wDataWord:=awBusDataToVTEM[0], xError=> );							// Valve Mode = 63
			fbwritevaluetoword(iValue:=0, iStartBit:=6, iEndBit:=7, wDataWord:=awBusDataToVTEM[0], xError=> );							// 0 (unused)
			fbwritevaluetoword(iValue:=0, iStartBit:=8, iEndBit:=12, wDataWord:=awBusDataToVTEM[0], xError=> );							// Channel = 0 (ignored)
			fbwritevaluetoword(iValue:=3, iStartBit:=13, iEndBit:=15, wDataWord:=awBusDataToVTEM[0], xError=> );						// Transfer Control = 3 (Exit transfer mode)
			fbwritevaluetoword(iValue:=0, iStartBit:=0, iEndBit:=7, wDataWord:=awBusDataToVTEM[1], xError=> );							// Addressed Target = 0 (ignored)
			fbwritevaluetoword(iValue:=0, iStartBit:=8, iEndBit:=15, wDataWord:=awBusDataToVTEM[1], xError=> );							// Index = 0 (ignored)
			fbwritevaluetoword(iValue:=0, iStartBit:=0, iEndBit:=15, wDataWord:=awBusDataToVTEM[2], xError=> );							// Value = 0 (ignored)
			
		6:	// STOP RUNNING MOTION APP
			fbwritevaluetoword(iValue:=61, iStartBit:=0, iEndBit:=5, wDataWord:=awBusDataToVTEM[0], xError=> );							// Valve Mode = 61 (stop)
			fbwritevaluetoword(iValue:=0, iStartBit:=6, iEndBit:=7, wDataWord:=awBusDataToVTEM[0], xError=> );							// App Control = 0 (unused)
			fbwritevaluetoword(iValue:=0, iStartBit:=8, iEndBit:=15, wDataWord:=awBusDataToVTEM[0], xError=> );							// App Option = 0 (unused)
			fbwritevaluetoword(iValue:=0, iStartBit:=0, iEndBit:=15, wDataWord:=awBusDataToVTEM[1], xError=> );							// Setpoint Value 1 = 0 (unused)
			fbwritevaluetoword(iValue:=0, iStartBit:=0, iEndBit:=15, wDataWord:=awBusDataToVTEM[2], xError=> );							// Setpoint Value 2 = 0 (unused)
		
		30:	// RUN FB_UPLOADMULTIPLEPARAMETERS
			fbuploadMultipleParameters(
				awBusDataFromVTEM:= awBusDataFromVTEM, 
				awBusDataToVTEM:= awBusDataToVTEM, 
				xExecute:= TRUE, 
				iResponse=> , 
				iCurrentValue=> , 
				xUploadDone=> , 
				xUploadError=> , 
				aTransferPackages:= aTransferPackages);

		40:	// RESET FB_UPLOADMULTIPLEPARAMETERS
			fbuploadMultipleParameters(
				awBusDataFromVTEM:= awBusDataFromVTEM, 
				awBusDataToVTEM:= awBusDataToVTEM, 
				xExecute:= FALSE, 
				iResponse=> , 
				iCurrentValue=> , 
				xUploadDone=> , 
				xUploadError=> , 
				aTransferPackages:= aTransferPackages);
	END_CASE
//-----------------------------------------------------------------------------------------------------------

END_FUNCTION_BLOCK

// Transfermode/specific_MA_config/FB_Read_config_MA_06
/// This function block can be used to upload the configuration of Motion App 6 ("ECO drive").
/// The specific parameters of this Motion App are the outputs of this FB
/// The function block uses the transfer mode to read this configuration from the Motion Terminal
/// and indicates the state of the upload process at the output iResponse.

FUNCTION_BLOCK FB_Read_config_MA_06
VAR_INPUT
	awBusDataFromVTEM 				: ARRAY [0..2] OF WORD;		// array of 3 words of process data received from the Motion Terminal
END_VAR
	
VAR_IN_OUT
	awBusDataToVTEM 				: ARRAY [0..2] OF WORD; 	// array of 3 words of process data sent to the Motion Terminal
END_VAR

VAR_INPUT
	xExecute 						: BOOL; 					// rising edge starts the reading process, falling edge resets the function block after reading is done
	xAbort							: BOOL;						// rising edge aborts the reading process
	iParameterSet					: INT := 1; 				// the parameter set to be read from, 1 by default
END_VAR                     		

VAR_OUTPUT                  		
	// system parameters
		iInPortRetracted			: INT;						// Sensor port for detection of end position at pressurisation of outlet port 2 (retracted), value is number of the slot (beginning from 0 and including valve slots) * 10 + number of the port
		iInPortAdvanced				: INT;						// Sensor port for detection of end position at pressurisation of outlet port 4 (advanced), value is number of the slot (beginning from 0 and including valve slots) * 10 + number of the port
		
	// function block response
		iResponse 					: eTransferResponse; 		// returns the status of the upload process
		xBusy						: BOOL;						// TRUE as long as the upload process is running
		xDone 						: BOOL; 					// indicates whether the upload was successfull
		xError 						: BOOL; 					// indicates whether an error occurred during the transfer
		xAborted					: BOOL;						// TRUE if the function block was canceled by xAbort	
END_VAR

VAR
	iState							: INT := 10;
	xStateChange					: BOOL;
	iCommandNumber					: INT;
	xFirstCycle						: BOOL := TRUE;				// indicator for the first cycle of the function block
	iParameterSetFC					: INT;						// value on input iParameterSet during first cycle
	
	aTransferPackages				: ARRAY [0..100] OF stTransferPackage;
	fbreadbitsfromword				: FB_Read_Bits_From_Word;
	fbuploadMultipleParameters 		: FB_Upload_Multiple_Parameters;
	fbWriteValueToWord 				: FB_Write_Value_To_Word;

	iCounterResetArray				: INT;

	iCurrentValveMode				: INT;						//
END_VAR

(*****************************************************************************************************

Festo SE & Co. KG, Esslingen
Copyright (c) 2021. All rights reserved.

Product:            Motion Terminal VTEM
Description:        Function Block to upload the parameters for Motion App 6 from the Motion Terminal

Object version:     2.00
Last change:        2021-07
======================================================================================================
                                       H I S T O R Y
======================================================================================================
Version:            2.00
Date:               2021-07
Change/Activity:    - created (#3872357)
Release:            3.5.7.237 (CODESYS 3.5.7.2, Lib version 3.7)
Author:             JEBU
======================================================================================================

*****************************************************************************************************)

// pre-check of the value for the parameter set
	IF xExecute = TRUE AND (iParameterSet < 1 OR iParameterSet > 5) THEN		// invalid input for the parameter set
		xDone := FALSE; 
		xError := TRUE; 
		iResponse := eTransferResponse.invalid_ParameterSet;
		xStateChange := TRUE;
		iState := 70;	// ERROR
	END_IF
//-----------------------------------------------------------------------------------------------------------

// check if iParameterSet was changed
	IF xExecute = TRUE AND xFirstCycle = TRUE THEN
		xFirstCycle := FALSE;
		iParameterSetFC := iParameterSet;
	END_IF
	
	IF xExecute = TRUE AND iParameterSet <> iParameterSetFC THEN
		xStateChange := TRUE;
		iState := 70;
		iResponse := eTransferResponse.FB_needs_rising_edge_xExecute;
	END_IF
//-----------------------------------------------------------------------------------------------------------

// WRITE PARAMETER INDICES INTO ARRAY
	//iInPortRetract
		aTransferPackages[0].iChannel := iParameterSet;
		aTransferPackages[0].iAddressedTarget := 6;
		aTransferPackages[0].iIndex := 70;
	
	//iInPortAdvanced
		aTransferPackages[1].iChannel := iParameterSet;
		aTransferPackages[1].iAddressedTarget := 6;
		aTransferPackages[1].iIndex := 71;
	
	// define end of parameter list to be uploaded by setting all variables to 0 (end criterion for FB_Upload_Multiple_Parameters)
		aTransferPackages[2].iChannel := 0;
		aTransferPackages[2].iAddressedTarget := 0;
		aTransferPackages[2].iIndex := 0;
//-----------------------------------------------------------------------------------------------------------

// Read the current status of the the motion terminal
	fbreadbitsfromword(wData:= awBusDataFromVTEM[0], iStartBit:=0, iEndBit:= 5, iValue=> iCurrentValveMode, xError=> );				// read current valve mode
//-----------------------------------------------------------------------------------------------------------

// Transition: Aborting condition when xAbort is TRUE in all States except "IDLE" , "ABORTING" and "RESETTING"
	IF xAbort = TRUE AND NOT(iState = 10 AND xExecute = FALSE) AND iState <> 80 AND iState <> 100 THEN
		xStateChange := TRUE;	// Leaving current state
		iState := 80;	// Choosing next state, here: ABORTING
	END_IF
//-----------------------------------------------------------------------------------------------------------

// local state machine
	CASE iState OF
		10:	// IDLE
			// code that is executed only in the first cycle of this state
				IF xStateChange = TRUE THEN
					xStateChange := FALSE;
					iResponse := eTransferResponse.ready_for_new_transfer;
					xDone := FALSE;
					xError := FALSE;
					xBusy := FALSE;
					xAborted := FALSE;
				END_IF
			//-----------------------------------------------------------------------------------------------------------
			
			// code that is repeated every cycle in this state
				iCommandNumber := 0;
			//-----------------------------------------------------------------------------------------------------------
			
			// Transition
			IF xExecute = TRUE THEN
				xStateChange := TRUE;
				iState := 20;
			END_IF
			//-----------------------------------------------------------------------------------------------------------
		
		20:	// RESETTING VALVE MODE TO 61
			// code that is executed only in the first cycle of this state
				IF xStateChange = TRUE THEN
					xStateChange := FALSE;
					iResponse := eTransferResponse.preparing_transfer;
					xDone := FALSE;
					xError := FALSE;
					xBusy := TRUE;
					xAborted := FALSE;
				END_IF
			//-----------------------------------------------------------------------------------------------------------
			
			// code that is repeated every cycle in this state	
				IF iCurrentValveMode = 63 THEN
					iCommandNumber := 5;	// exit transfer mode
				ELSIF iCurrentValveMode <> 61 AND iCurrentValveMode <> 63 THEN
					iCommandNumber := 6;	// stop running motion apps
				END_IF 
			//-----------------------------------------------------------------------------------------------------------
			
			// Transition
				IF iCurrentValveMode = 61 THEN
					xStateChange := TRUE;	// Leave this state
					iState := 30;
					iCommandNumber := 30;			
				END_IF
			//-----------------------------------------------------------------------------------------------------------
		
		30:	// READING PARAMETER VALUES
			// code that is executed only in the first cycle of this state
				IF xStateChange = TRUE THEN
					xStateChange := FALSE;
					iResponse := eTransferResponse.transferring;
					xDone := FALSE;
					xError := FALSE;
					xBusy := TRUE;
					xAborted := FALSE;
				END_IF
			//-----------------------------------------------------------------------------------------------------------
			
			// code that is repeated every cycle in this state
				iCommandNumber := 30;		// read parameter values
			//-----------------------------------------------------------------------------------------------------------
			
			// Transition
				IF fbuploadMultipleParameters.xExecute = TRUE AND fbuploadMultipleParameters.xUploadDone = TRUE AND fbuploadMultipleParameters.xUploadError = FALSE THEN	// Upload Done
					xStateChange := TRUE;
					iState := 40;	// Write parameter values to outputs
				ELSIF fbuploadMultipleParameters.xExecute = TRUE AND fbuploadMultipleParameters.xUploadDone = FALSE AND fbuploadMultipleParameters.xUploadError = TRUE THEN	// Error during update
					xStateChange := TRUE;
					iState := 70;	// ERROR
					iResponse := fbuploadMultipleParameters.iResponse;
				END_IF
			//-----------------------------------------------------------------------------------------------------------
		
		40:	// WRITE PARAMETER VALUES TO OUTPUTS
			// code that is executed only in the first cycle of this state
				IF xStateChange = TRUE THEN
					xStateChange := FALSE;
					iResponse := eTransferResponse.transferring;
					xDone := FALSE;
					xError := FALSE;
					xBusy := TRUE;
					xAborted := FALSE;
				END_IF
			//-----------------------------------------------------------------------------------------------------------
			
			// code that is repeated every cycle in this state
				iInPortRetracted	:= aTransferPackages[0].iTransferValue;
				iInPortAdvanced		:= aTransferPackages[1].iTransferValue;
			//-----------------------------------------------------------------------------------------------------------
			
			// Transition
				xStateChange := TRUE;
				iState := 50;
				iCommandNumber := 40;
			//-----------------------------------------------------------------------------------------------------------
		
		50:	// DONE
			// code that is executed only in the first cycle of this state
				IF xStateChange = TRUE THEN
					xStateChange := FALSE;
					iResponse := eTransferResponse.transfer_successful;
					xDone := TRUE;
					xError := FALSE;
					xBusy := FALSE;
					xAborted := FALSE;
				END_IF
			//-----------------------------------------------------------------------------------------------------------
			
			// code that is repeated every cycle in this state	
				IF fbuploadMultipleParameters.xExecute = FALSE  AND fbuploadMultipleParameters.xUploadDone = FALSE AND fbuploadMultipleParameters.xUploadError = FALSE AND iCurrentValveMode = 63 THEN		//FB_UploadMultipleParameters was reset
					iCommandNumber := 5;	// exit transfer mode
				END_IF
			//-----------------------------------------------------------------------------------------------------------
			
			// Transition
				IF fbuploadMultipleParameters.xExecute = FALSE  AND fbuploadMultipleParameters.xUploadDone = FALSE AND fbuploadMultipleParameters.xUploadError = FALSE AND xExecute = FALSE THEN
					xStateChange := TRUE;
					iState := 100;
				END_IF
			//-----------------------------------------------------------------------------------------------------------
			
		70:	// ERROR
			// code that is executed only in the first cycle of this state
				IF xStateChange = TRUE THEN
					xStateChange := FALSE;
					//iResponse := eTransferResponse.communication_failed;	// set within the transition of the last state
					xDone := FALSE;
					xError := TRUE;
					xBusy := FALSE;
					xAborted := FALSE;
				END_IF
			//-----------------------------------------------------------------------------------------------------------
			
			// code that is repeated every cycle in this state	
			//-----------------------------------------------------------------------------------------------------------
			
			// Transition
				IF xExecute = FALSE AND xAbort = FALSE THEN
					xStateChange := TRUE;
					iState := 100;
				END_IF
			//-----------------------------------------------------------------------------------------------------------
			
		80:	// ABORTING
			// code that is executed only in the first cycle of this state
				IF xStateChange = TRUE THEN
					xStateChange := FALSE;
					iResponse := eTransferResponse.aborting;
					xBusy := FALSE;
					xDone := FALSE;
					xError := FALSE;
					xAborted := TRUE;
				END_IF
			//-----------------------------------------------------------------------------------------------------------
			
			// code that is repeated every cycle in this state
				IF iCurrentValveMode = 63 THEN
					iCommandNumber := 5;	// exit transfer mode
				ELSIF iCurrentValveMode <> 61 AND iCurrentValveMode <> 63 THEN
					iCommandNumber := 6;	// stop running motion apps
				ELSE
					iCommandNumber := 0; 
				END_IF
			//-----------------------------------------------------------------------------------------------------------
			
			// Transition
				IF xAbort = FALSE AND xExecute = FALSE AND iCurrentValveMode = 61 THEN
					xStateChange := TRUE;
					iState := 100;
				END_IF
			//-----------------------------------------------------------------------------------------------------------

		100:	// RESETTING FUNCTION BLOCK AND VALVE
			// code that is executed only in the first cycle of this state
				IF xStateChange = TRUE THEN
					xStateChange := FALSE;
					iResponse := eTransferResponse.resetting;
					xDone := FALSE;
					xError := FALSE;
					xBusy := FALSE;
					xAborted := FALSE;
				END_IF
			//-----------------------------------------------------------------------------------------------------------
			
			// code that is repeated every cycle in this state	
				IF iCurrentValveMode = 63 THEN
					iCommandNumber := 5;	// exit transfer mode
				ELSIF iCurrentValveMode <> 61 AND iCurrentValveMode <> 63 THEN
					iCommandNumber := 6;	// stop running motion apps
				END_IF
				
				// reset funktion block fbreadmultipleparameters
				// not done via command number because this is used to reset valve
					fbuploadMultipleParameters(
						awBusDataFromVTEM:= awBusDataFromVTEM, 
						awBusDataToVTEM:= awBusDataToVTEM, 
						xExecute:= FALSE, 
						iResponse=> , 
						iCurrentValue=> , 
						xUploadDone=> , 
						xUploadError=> , 
						aTransferPackages:= aTransferPackages);
				
				// reset parameter outputs
					iParameterSet				:= 1;

					iInPortRetracted	:= 0;
					iInPortAdvanced		:= 0;
				
				// reset parameter array
					FOR iCounterResetArray := 0 TO 100 BY 1 DO
						aTransferPackages[iCounterResetArray].iChannel := 0;
						aTransferPackages[iCounterResetArray].iAddressedTarget := 0;
						aTransferPackages[iCounterResetArray].iIndex := 0;
						aTransferPackages[iCounterResetArray].iTransferValue := 0;
					END_FOR
					
					iCounterResetArray := 0;
					xFirstCycle := TRUE;
			//-----------------------------------------------------------------------------------------------------------
			
			// Transition
				IF iCurrentValveMode = 61 THEN
					iCommandNumber := 6; // Last command to send before the FB is in IDLE
					xStateChange := TRUE;
					iState := 10;
				END_IF
			//-----------------------------------------------------------------------------------------------------------
			
	END_CASE
//-----------------------------------------------------------------------------------------------------------

// Command section
	CASE iCommandNumber OF
		0:	// IDLE
			;
		
		5:	// EXIT TRANSFER MODE
			fbwritevaluetoword(iValue:=63, iStartBit:=0, iEndBit:=5, wDataWord:=awBusDataToVTEM[0], xError=> );							// Valve Mode = 63
			fbwritevaluetoword(iValue:=0, iStartBit:=6, iEndBit:=7, wDataWord:=awBusDataToVTEM[0], xError=> );							// 0 (unused)
			fbwritevaluetoword(iValue:=0, iStartBit:=8, iEndBit:=12, wDataWord:=awBusDataToVTEM[0], xError=> );							// Channel = 0 (ignored)
			fbwritevaluetoword(iValue:=3, iStartBit:=13, iEndBit:=15, wDataWord:=awBusDataToVTEM[0], xError=> );						// Transfer Control = 3 (Exit transfer mode)
			fbwritevaluetoword(iValue:=0, iStartBit:=0, iEndBit:=7, wDataWord:=awBusDataToVTEM[1], xError=> );							// Addressed Target = 0 (ignored)
			fbwritevaluetoword(iValue:=0, iStartBit:=8, iEndBit:=15, wDataWord:=awBusDataToVTEM[1], xError=> );							// Index = 0 (ignored)
			fbwritevaluetoword(iValue:=0, iStartBit:=0, iEndBit:=15, wDataWord:=awBusDataToVTEM[2], xError=> );							// Value = 0 (ignored)
			
		6:	// STOP RUNNING MOTION APP
			fbwritevaluetoword(iValue:=61, iStartBit:=0, iEndBit:=5, wDataWord:=awBusDataToVTEM[0], xError=> );							// Valve Mode = 61 (stop)
			fbwritevaluetoword(iValue:=0, iStartBit:=6, iEndBit:=7, wDataWord:=awBusDataToVTEM[0], xError=> );							// App Control = 0 (unused)
			fbwritevaluetoword(iValue:=0, iStartBit:=8, iEndBit:=15, wDataWord:=awBusDataToVTEM[0], xError=> );							// App Option = 0 (unused)
			fbwritevaluetoword(iValue:=0, iStartBit:=0, iEndBit:=15, wDataWord:=awBusDataToVTEM[1], xError=> );							// Setpoint Value 1 = 0 (unused)
			fbwritevaluetoword(iValue:=0, iStartBit:=0, iEndBit:=15, wDataWord:=awBusDataToVTEM[2], xError=> );							// Setpoint Value 2 = 0 (unused)
		
		30:	// RUN FB_UPLOADMULTIPLEPARAMETERS
			fbuploadMultipleParameters(
				awBusDataFromVTEM:= awBusDataFromVTEM, 
				awBusDataToVTEM:= awBusDataToVTEM, 
				xExecute:= TRUE, 
				iResponse=> , 
				iCurrentValue=> , 
				xUploadDone=> , 
				xUploadError=> , 
				aTransferPackages:= aTransferPackages);

		40:	// RESET FB_UPLOADMULTIPLEPARAMETERS
			fbuploadMultipleParameters(
				awBusDataFromVTEM:= awBusDataFromVTEM, 
				awBusDataToVTEM:= awBusDataToVTEM, 
				xExecute:= FALSE, 
				iResponse=> , 
				iCurrentValue=> , 
				xUploadDone=> , 
				xUploadError=> , 
				aTransferPackages:= aTransferPackages);
	END_CASE
//-----------------------------------------------------------------------------------------------------------

END_FUNCTION_BLOCK

// Transfermode/specific_MA_config/FB_Read_config_MA_07
/// This function block can be used to upload the configuration of Motion App 7 ("Presetting of travel time").
/// The specific parameters of this Motion App are the outputs of this FB
/// The function block uses the transfer mode to read this configuration from the Motion Terminal
/// and indicates the state of the upload process at the output iResponse.

FUNCTION_BLOCK FB_Read_config_MA_07
VAR_INPUT
	awBusDataFromVTEM 				: ARRAY [0..2] OF WORD;		// array of 3 words of process data received from the Motion Terminal
END_VAR
	
VAR_IN_OUT
	awBusDataToVTEM 				: ARRAY [0..2] OF WORD; 	// array of 3 words of process data sent to the Motion Terminal
END_VAR

VAR_INPUT
	xExecute 						: BOOL; 					// rising edge starts the reading process, falling edge resets the function block after reading is done
	xAbort							: BOOL;						// rising edge aborts the reading process
	iParameterSet					: INT := 1; 				// the parameter set to be read from, 1 by default
END_VAR                     		

VAR_OUTPUT                  		
	// system parameters                 		                        	
		iTubingLengthAt2 			: INT; 						// length of the tubing connected to outlet port 2 of the valve [1 digit = 1 mm]
 		iTubingLengthAt4 			: INT;						// length of the tubing connected to outlet port 4 of the valve [1 digit = 1 mm]
 		iTubingInnerDiameterAt2		: INT;  					// inner diameter of the tubing connected to outlet port 2 of the valve [1 digit = 0.01 mm]
 		iTubingInnerDiameterAt4		: INT;						// inner diameter of the tubing connected to outlet port 4 of the valve [1 digit = 0.01 mm]
 		iDriveType 					: INT;						// type of the drive/cylinder/... that is to be operated by the valve ->  see list of drive types at support portal (www.festo.com/sp/)
 		iDriveStroke 				: INT; 						// stroke of the drive/cylinder/... that is to be operated by the valve [1 digit = 1 mm for linear drives, 1 digit = 1° for rotary drives]
		iInstallationPositionDrive 	: INT;  	 				// inclination of the cylinder with reference to a horizontal installation position [1 digit = 0.01°, positive values = advancing upwards]
		iInPortRetracted			: INT;						// Sensor port for detection of end position at pressurisation of outlet port 2 (retracted), value is number of the slot (beginning from 0 and including valve slots) * 10 + number of the port
		iInPortAdvanced				: INT;						// Sensor port for detection of end position at pressurisation of outlet port 4 (advanced), value is number of the slot (beginning from 0 and including valve slots) * 10 + number of the port
	                                                        	
	// application parameters                               	
		iLoadRetracting 			: INT;						// mass that is to be moved by the drive when retracting ((2) pressurised) [1 digit = 0.01 kg]
 		iLoadAdvancing 				: INT; 						// mass that is to be moved by the drive when advancing ((4) pressurised) [1 digit = 0.01 kg]
		iMomentOfInertiaRetracting	: INT;						// Moment of inertia during for swivel drives when retratcting ((2) pressirised) [1 digit = 1 kg cm³]
		iMomentOfInertiaAdvancing	: INT;						// Moment of inertia during for swivel drives when advancing ((4) pressirised) [1 digit = 1 kg cm³]
		iTravelTimeRetracting 		: INT;						// preset travel time from one end position to the other when retracting ((2) pressurised) [1 digit = 0.01 s]
		iTravelTimeAdvancing 		: INT; 						// preset travel time from one end position to the other when advancing ((4) pressurised) [1 digit = 0.01 s]
		iSoftStartFunction			: INT;						// flag to enable or disable the iSoftStartFunction; 0 = disabled, 1 = enabled
		
	// function block response
		iResponse 					: eTransferResponse; 		// returns the status of the upload process
		xBusy						: BOOL;						// TRUE as long as the upload process is running
		xDone 						: BOOL; 					// indicates whether the upload was successfull
		xError 						: BOOL; 					// indicates whether an error occurred during the transfer
		xAborted					: BOOL;						// TRUE if the function block was canceled by xAbort	
END_VAR

VAR
	iState							: INT := 10;
	xStateChange					: BOOL;
	iCommandNumber					: INT;
	xFirstCycle						: BOOL := TRUE;				// indicator for the first cycle of the function block
	iParameterSetFC					: INT;						// value on input iParameterSet during first cycle
	
	aTransferPackages				: ARRAY [0..100] OF stTransferPackage;
	fbreadbitsfromword				: FB_Read_Bits_From_Word;
	fbuploadMultipleParameters 		: FB_Upload_Multiple_Parameters;
	fbWriteValueToWord 				: FB_Write_Value_To_Word;

	iCounterResetArray				: INT;

	iCurrentValveMode				: INT;						//
END_VAR

(*****************************************************************************************************

Festo SE & Co. KG, Esslingen
Copyright (c) 2021. All rights reserved.

Product:            Motion Terminal VTEM
Description:        Function Block to upload the parameters for Motion App 7 from the Motion Terminal

Object version:     2.00
Last change:        2021-07
======================================================================================================
                                       H I S T O R Y
======================================================================================================
Version:            2.00
Date:               2021-07
Change/Activity:    - created (#3872357)
Release:            3.5.7.237 (CODESYS 3.5.7.2, Lib version 3.7)
Author:             JEBU
======================================================================================================

*****************************************************************************************************)

// pre-check of the value for the parameter set
	IF xExecute = TRUE AND (iParameterSet < 1 OR iParameterSet > 5) THEN		// invalid input for the parameter set
		xDone := FALSE; 
		xError := TRUE; 
		iResponse := eTransferResponse.invalid_ParameterSet;
		xStateChange := TRUE;
		iState := 70;	// ERROR
	END_IF
//-----------------------------------------------------------------------------------------------------------

// check if iParameterSet was changed
	IF xExecute = TRUE AND xFirstCycle = TRUE THEN
		xFirstCycle := FALSE;
		iParameterSetFC := iParameterSet;
	END_IF
	
	IF xExecute = TRUE AND iParameterSet <> iParameterSetFC THEN
		xStateChange := TRUE;
		iState := 70;
		iResponse := eTransferResponse.FB_needs_rising_edge_xExecute;
	END_IF
//-----------------------------------------------------------------------------------------------------------

// WRITE PARAMETER INDICES INTO ARRAY
	//iTubingLengthAt2
		aTransferPackages[0].iChannel := iParameterSet;
		aTransferPackages[0].iAddressedTarget := 7;
		aTransferPackages[0].iIndex := 12;
		
	//iTubingLengthAt4
		aTransferPackages[1].iChannel := iParameterSet;
		aTransferPackages[1].iAddressedTarget := 7;
		aTransferPackages[1].iIndex := 13;
		
	//iTubingInnerDiameterAt2
		aTransferPackages[2].iChannel := iParameterSet;
		aTransferPackages[2].iAddressedTarget := 7;
		aTransferPackages[2].iIndex := 14;
		
	//iTubingInnerDiameterAt4
		aTransferPackages[3].iChannel := iParameterSet;
		aTransferPackages[3].iAddressedTarget := 7;
		aTransferPackages[3].iIndex := 15;
		
	//iDriveType
		aTransferPackages[4].iChannel := iParameterSet;
		aTransferPackages[4].iAddressedTarget := 7;
		aTransferPackages[4].iIndex := 20;
		
	//iDriveStroke
		aTransferPackages[5].iChannel := iParameterSet;
		aTransferPackages[5].iAddressedTarget := 7;
		aTransferPackages[5].iIndex := 21;
		
	//iInstallationPositionDrive
		aTransferPackages[6].iChannel := iParameterSet;
		aTransferPackages[6].iAddressedTarget := 7;
		aTransferPackages[6].iIndex := 60;
		
	//iLoadRetracting
		aTransferPackages[7].iChannel := iParameterSet;
		aTransferPackages[7].iAddressedTarget := 7;
		aTransferPackages[7].iIndex := 100;
		
	//iLoadAdvancing
		aTransferPackages[8].iChannel := iParameterSet;
		aTransferPackages[8].iAddressedTarget := 7;
		aTransferPackages[8].iIndex := 101;
		
	//iMomentOfInertiaRetracting
		aTransferPackages[9].iChannel := iParameterSet;
		aTransferPackages[9].iAddressedTarget := 7;
		aTransferPackages[9].iIndex := 102;
	
	//iMomentOfInertiaAdvancing
		aTransferPackages[10].iChannel := iParameterSet;
		aTransferPackages[10].iAddressedTarget := 7;
		aTransferPackages[10].iIndex := 103;

	//iTravelTimeRetracting
		aTransferPackages[11].iChannel := iParameterSet;
		aTransferPackages[11].iAddressedTarget := 7;
		aTransferPackages[11].iIndex := 120;
	
	//iTravelTimeAdvancing
		aTransferPackages[12].iChannel := iParameterSet;
		aTransferPackages[12].iAddressedTarget := 7;
		aTransferPackages[12].iIndex := 121;
	
	//iSoftStartFunction
		aTransferPackages[13].iChannel := iParameterSet;
		aTransferPackages[13].iAddressedTarget := 7;
		aTransferPackages[13].iIndex := 222;
	
	//iInPortRetract
		aTransferPackages[14].iChannel := iParameterSet;
		aTransferPackages[14].iAddressedTarget := 7;
		aTransferPackages[14].iIndex := 70;
	
	//iInPortRetract
		aTransferPackages[15].iChannel := iParameterSet;
		aTransferPackages[15].iAddressedTarget := 7;
		aTransferPackages[15].iIndex := 71;
	
	// define end of parameter list to be uploaded by setting all variables to 0 (end criterion for FB_Upload_Multiple_Parameters)
		aTransferPackages[16].iChannel := 0;
		aTransferPackages[16].iAddressedTarget := 0;
		aTransferPackages[16].iIndex := 0;
//-----------------------------------------------------------------------------------------------------------

// Read the current status of the the motion terminal
	fbreadbitsfromword(wData:= awBusDataFromVTEM[0], iStartBit:=0, iEndBit:= 5, iValue=> iCurrentValveMode, xError=> );				// read current valve mode
//-----------------------------------------------------------------------------------------------------------

// Transition: Aborting condition when xAbort is TRUE in all States except "IDLE" , "ABORTING" and "RESETTING"
	IF xAbort = TRUE AND NOT(iState = 10 AND xExecute = FALSE) AND iState <> 80 AND iState <> 100 THEN
		xStateChange := TRUE;	// Leaving current state
		iState := 80;	// Choosing next state, here: ABORTING
	END_IF
//-----------------------------------------------------------------------------------------------------------

// local state machine
	CASE iState OF
		10:	// IDLE
			// code that is executed only in the first cycle of this state
				IF xStateChange = TRUE THEN
					xStateChange := FALSE;
					iResponse := eTransferResponse.ready_for_new_transfer;
					xDone := FALSE;
					xError := FALSE;
					xBusy := FALSE;
					xAborted := FALSE;
				END_IF
			//-----------------------------------------------------------------------------------------------------------
			
			// code that is repeated every cycle in this state
				iCommandNumber := 0;
			//-----------------------------------------------------------------------------------------------------------
			
			// Transition
			IF xExecute = TRUE THEN
				xStateChange := TRUE;
				iState := 20;
			END_IF
			//-----------------------------------------------------------------------------------------------------------
		
		20:	// RESETTING VALVE MODE TO 61
			// code that is executed only in the first cycle of this state
				IF xStateChange = TRUE THEN
					xStateChange := FALSE;
					iResponse := eTransferResponse.preparing_transfer;
					xDone := FALSE;
					xError := FALSE;
					xBusy := TRUE;
					xAborted := FALSE;
				END_IF
			//-----------------------------------------------------------------------------------------------------------
			
			// code that is repeated every cycle in this state	
				IF iCurrentValveMode = 63 THEN
					iCommandNumber := 5;	// exit transfer mode
				ELSIF iCurrentValveMode <> 61 AND iCurrentValveMode <> 63 THEN
					iCommandNumber := 6;	// stop running motion apps
				END_IF 
			//-----------------------------------------------------------------------------------------------------------
			
			// Transition
				IF iCurrentValveMode = 61 THEN
					xStateChange := TRUE;	// Leave this state
					iState := 30;
					iCommandNumber := 30;			
				END_IF
			//-----------------------------------------------------------------------------------------------------------
		
		30:	// READING PARAMETER VALUES
			// code that is executed only in the first cycle of this state
				IF xStateChange = TRUE THEN
					xStateChange := FALSE;
					iResponse := eTransferResponse.transferring;
					xDone := FALSE;
					xError := FALSE;
					xBusy := TRUE;
					xAborted := FALSE;
				END_IF
			//-----------------------------------------------------------------------------------------------------------
			
			// code that is repeated every cycle in this state
				iCommandNumber := 30;		// read parameter values
			//-----------------------------------------------------------------------------------------------------------
			
			// Transition
				IF fbuploadMultipleParameters.xExecute = TRUE AND fbuploadMultipleParameters.xUploadDone = TRUE AND fbuploadMultipleParameters.xUploadError = FALSE THEN	// Upload Done
					xStateChange := TRUE;
					iState := 40;	// Write parameter values to outputs
				ELSIF fbuploadMultipleParameters.xExecute = TRUE AND fbuploadMultipleParameters.xUploadDone = FALSE AND fbuploadMultipleParameters.xUploadError = TRUE THEN	// Error during update
					xStateChange := TRUE;
					iState := 70;	// ERROR
					iResponse := fbuploadMultipleParameters.iResponse;
				END_IF
			//-----------------------------------------------------------------------------------------------------------
		
		40:	// WRITE PARAMETER VALUES TO OUTPUTS
			// code that is executed only in the first cycle of this state
				IF xStateChange = TRUE THEN
					xStateChange := FALSE;
					iResponse := eTransferResponse.transferring;
					xDone := FALSE;
					xError := FALSE;
					xBusy := TRUE;
					xAborted := FALSE;
				END_IF
			//-----------------------------------------------------------------------------------------------------------
			
			// code that is repeated every cycle in this state
				iTubingLengthAt2			:= aTransferPackages[0].iTransferValue;
				iTubingLengthAt4			:= aTransferPackages[1].iTransferValue;
				iTubingInnerDiameterAt2		:= aTransferPackages[2].iTransferValue;
				iTubingInnerDiameterAt4		:= aTransferPackages[3].iTransferValue;
				iDriveType					:= aTransferPackages[4].iTransferValue;
				iDriveStroke				:= aTransferPackages[5].iTransferValue;
				iInstallationPositionDrive	:= aTransferPackages[6].iTransferValue;
				iLoadRetracting				:= aTransferPackages[7].iTransferValue;
				iLoadAdvancing				:= aTransferPackages[8].iTransferValue;
				iMomentOfInertiaRetracting	:= aTransferPackages[9].iTransferValue;
				iMomentOfInertiaAdvancing	:= aTransferPackages[10].iTransferValue;
				iTravelTimeRetracting		:= aTransferPackages[11].iTransferValue;
				iTravelTimeAdvancing		:= aTransferPackages[12].iTransferValue;
				iSoftStartFunction			:= aTransferPackages[13].iTransferValue;
				iInPortRetracted			:= aTransferPackages[14].iTransferValue;
				iInPortAdvanced				:= aTransferPackages[15].iTransferValue;
			//-----------------------------------------------------------------------------------------------------------
			
			// Transition
				xStateChange := TRUE;
				iState := 50;
				iCommandNumber := 40;
			//-----------------------------------------------------------------------------------------------------------
		
		50:	// DONE
			// code that is executed only in the first cycle of this state
				IF xStateChange = TRUE THEN
					xStateChange := FALSE;
					iResponse := eTransferResponse.transfer_successful;
					xDone := TRUE;
					xError := FALSE;
					xBusy := FALSE;
					xAborted := FALSE;
				END_IF
			//-----------------------------------------------------------------------------------------------------------
			
			// code that is repeated every cycle in this state	
				IF fbuploadMultipleParameters.xExecute = FALSE  AND fbuploadMultipleParameters.xUploadDone = FALSE AND fbuploadMultipleParameters.xUploadError = FALSE AND iCurrentValveMode = 63 THEN		//FB_UploadMultipleParameters was reset
					iCommandNumber := 5;	// exit transfer mode
				END_IF
			//-----------------------------------------------------------------------------------------------------------
			
			// Transition
				IF fbuploadMultipleParameters.xExecute = FALSE  AND fbuploadMultipleParameters.xUploadDone = FALSE AND fbuploadMultipleParameters.xUploadError = FALSE AND xExecute = FALSE THEN
					xStateChange := TRUE;
					iState := 100;
				END_IF
			//-----------------------------------------------------------------------------------------------------------
			
		70:	// ERROR
			// code that is executed only in the first cycle of this state
				IF xStateChange = TRUE THEN
					xStateChange := FALSE;
					//iResponse := eTransferResponse.communication_failed;	// set within the transition of the last state
					xDone := FALSE;
					xError := TRUE;
					xBusy := FALSE;
					xAborted := FALSE;
				END_IF
			//-----------------------------------------------------------------------------------------------------------
			
			// code that is repeated every cycle in this state	
			//-----------------------------------------------------------------------------------------------------------
			
			// Transition
				IF xExecute = FALSE AND xAbort = FALSE THEN
					xStateChange := TRUE;
					iState := 100;
				END_IF
			//-----------------------------------------------------------------------------------------------------------
			
		80:	// ABORTING
			// code that is executed only in the first cycle of this state
				IF xStateChange = TRUE THEN
					xStateChange := FALSE;
					iResponse := eTransferResponse.aborting;
					xBusy := FALSE;
					xDone := FALSE;
					xError := FALSE;
					xAborted := TRUE;
				END_IF
			//-----------------------------------------------------------------------------------------------------------
			
			// code that is repeated every cycle in this state
				IF iCurrentValveMode = 63 THEN
					iCommandNumber := 5;	// exit transfer mode
				ELSIF iCurrentValveMode <> 61 AND iCurrentValveMode <> 63 THEN
					iCommandNumber := 6;	// stop running motion apps
				ELSE
					iCommandNumber := 0; 
				END_IF
			//-----------------------------------------------------------------------------------------------------------
			
			// Transition
				IF xAbort = FALSE AND xExecute = FALSE AND iCurrentValveMode = 61 THEN
					xStateChange := TRUE;
					iState := 100;
				END_IF
			//-----------------------------------------------------------------------------------------------------------

		100:	// RESETTING FUNCTION BLOCK AND VALVE
			// code that is executed only in the first cycle of this state
				IF xStateChange = TRUE THEN
					xStateChange := FALSE;
					iResponse := eTransferResponse.resetting;
					xDone := FALSE;
					xError := FALSE;
					xBusy := FALSE;
					xAborted := FALSE;
				END_IF
			//-----------------------------------------------------------------------------------------------------------
			
			// code that is repeated every cycle in this state	
				IF iCurrentValveMode = 63 THEN
					iCommandNumber := 5;	// exit transfer mode
				ELSIF iCurrentValveMode <> 61 AND iCurrentValveMode <> 63 THEN
					iCommandNumber := 6;	// stop running motion apps
				END_IF
				
				// reset funktion block fbreadmultipleparameters
				// not done via command number because this is used to reset valve
					fbuploadMultipleParameters(
						awBusDataFromVTEM:= awBusDataFromVTEM, 
						awBusDataToVTEM:= awBusDataToVTEM, 
						xExecute:= FALSE, 
						iResponse=> , 
						iCurrentValue=> , 
						xUploadDone=> , 
						xUploadError=> , 
						aTransferPackages:= aTransferPackages);

				// reset parameter outputs
					iParameterSet				:= 1;

					iTubingLengthAt2			:= 0;
					iTubingLengthAt4			:= 0;
					iTubingInnerDiameterAt2		:= 0;
					iTubingInnerDiameterAt4		:= 0;
					iDriveType					:= 0;
					iDriveStroke				:= 0;
					iInstallationPositionDrive	:= 0;
					iLoadRetracting				:= 0;
					iLoadAdvancing				:= 0;
					iMomentOfInertiaRetracting	:= 0;
					iMomentOfInertiaAdvancing	:= 0;
					iTravelTimeRetracting		:= 0;
					iTravelTimeAdvancing		:= 0;
					iSoftStartFunction			:= 0;
					iInPortRetracted			:= 0;
					iInPortAdvanced				:= 0;
				
				// reset parameter array
					FOR iCounterResetArray := 0 TO 100 BY 1 DO
						aTransferPackages[iCounterResetArray].iChannel := 0;
						aTransferPackages[iCounterResetArray].iAddressedTarget := 0;
						aTransferPackages[iCounterResetArray].iIndex := 0;
						aTransferPackages[iCounterResetArray].iTransferValue := 0;
					END_FOR
					
					iCounterResetArray := 0;
					xFirstCycle := TRUE;
			//-----------------------------------------------------------------------------------------------------------
			
			// Transition
				IF iCurrentValveMode = 61 THEN
					iCommandNumber := 6; // Last command to send before the FB is in IDLE
					xStateChange := TRUE;
					iState := 10;
				END_IF
			//-----------------------------------------------------------------------------------------------------------
			
	END_CASE
//-----------------------------------------------------------------------------------------------------------

// Command section
	CASE iCommandNumber OF
		0:	// IDLE
			;
		
		5:	// EXIT TRANSFER MODE
			fbwritevaluetoword(iValue:=63, iStartBit:=0, iEndBit:=5, wDataWord:=awBusDataToVTEM[0], xError=> );							// Valve Mode = 63
			fbwritevaluetoword(iValue:=0, iStartBit:=6, iEndBit:=7, wDataWord:=awBusDataToVTEM[0], xError=> );							// 0 (unused)
			fbwritevaluetoword(iValue:=0, iStartBit:=8, iEndBit:=12, wDataWord:=awBusDataToVTEM[0], xError=> );							// Channel = 0 (ignored)
			fbwritevaluetoword(iValue:=3, iStartBit:=13, iEndBit:=15, wDataWord:=awBusDataToVTEM[0], xError=> );						// Transfer Control = 3 (Exit transfer mode)
			fbwritevaluetoword(iValue:=0, iStartBit:=0, iEndBit:=7, wDataWord:=awBusDataToVTEM[1], xError=> );							// Addressed Target = 0 (ignored)
			fbwritevaluetoword(iValue:=0, iStartBit:=8, iEndBit:=15, wDataWord:=awBusDataToVTEM[1], xError=> );							// Index = 0 (ignored)
			fbwritevaluetoword(iValue:=0, iStartBit:=0, iEndBit:=15, wDataWord:=awBusDataToVTEM[2], xError=> );							// Value = 0 (ignored)
			
		6:	// STOP RUNNING MOTION APP
			fbwritevaluetoword(iValue:=61, iStartBit:=0, iEndBit:=5, wDataWord:=awBusDataToVTEM[0], xError=> );							// Valve Mode = 61 (stop)
			fbwritevaluetoword(iValue:=0, iStartBit:=6, iEndBit:=7, wDataWord:=awBusDataToVTEM[0], xError=> );							// App Control = 0 (unused)
			fbwritevaluetoword(iValue:=0, iStartBit:=8, iEndBit:=15, wDataWord:=awBusDataToVTEM[0], xError=> );							// App Option = 0 (unused)
			fbwritevaluetoword(iValue:=0, iStartBit:=0, iEndBit:=15, wDataWord:=awBusDataToVTEM[1], xError=> );							// Setpoint Value 1 = 0 (unused)
			fbwritevaluetoword(iValue:=0, iStartBit:=0, iEndBit:=15, wDataWord:=awBusDataToVTEM[2], xError=> );							// Setpoint Value 2 = 0 (unused)
		
		30:	// RUN FB_UPLOADMULTIPLEPARAMETERS
			fbuploadMultipleParameters(
				awBusDataFromVTEM:= awBusDataFromVTEM, 
				awBusDataToVTEM:= awBusDataToVTEM, 
				xExecute:= TRUE, 
				iResponse=> , 
				iCurrentValue=> , 
				xUploadDone=> , 
				xUploadError=> , 
				aTransferPackages:= aTransferPackages);

		40:	// RESET FB_UPLOADMULTIPLEPARAMETERS
			fbuploadMultipleParameters(
				awBusDataFromVTEM:= awBusDataFromVTEM, 
				awBusDataToVTEM:= awBusDataToVTEM, 
				xExecute:= FALSE, 
				iResponse=> , 
				iCurrentValue=> , 
				xUploadDone=> , 
				xUploadError=> , 
				aTransferPackages:= aTransferPackages);
	END_CASE
//-----------------------------------------------------------------------------------------------------------

END_FUNCTION_BLOCK

// Transfermode/specific_MA_config/FB_Read_config_MA_08
/// This function block can be used to upload the configuration of Motion App 8 ("Selectable pressure level (ECO)").
/// The specific parameters of this Motion App are the outputs of this FB
/// The function block uses the transfer mode to read this configuration from the Motion Terminal
/// and indicates the state of the upload process at the output iResponse.

FUNCTION_BLOCK FB_Read_config_MA_08
VAR_INPUT
	awBusDataFromVTEM 				: ARRAY [0..2] OF WORD;		// array of 3 words of process data received from the Motion Terminal
END_VAR
	
VAR_IN_OUT
	awBusDataToVTEM 				: ARRAY [0..2] OF WORD; 	// array of 3 words of process data sent to the Motion Terminal
END_VAR

VAR_INPUT
	xExecute 						: BOOL; 					// rising edge starts the reading process, falling edge resets the function block after reading is done
	xAbort							: BOOL;						// rising edge aborts the reading process
	iParameterSet					: INT := 1; 				// the parameter set to be read from, 1 by default
END_VAR                     		

VAR_OUTPUT                  		
	// system parameters
		iTubingLengthAt2 			: INT; 						// length of the tubing connected to outlet port 2 of the valve [1 digit = 1 mm]
	 	iTubingLengthAt4 			: INT;						// length of the tubing connected to outlet port 4 of the valve [1 digit = 1 mm]
	 	iTubingInnerDiameterAt2		: INT;  					// inner diameter of the tubing connected to outlet port 2 of the valve [1 digit = 0.01 mm]
	 	iTubingInnerDiameterAt4		: INT;						// inner diameter of the tubing connected to outlet port 4 of the valve [1 digit = 0.01 mm]
	 	iDriveType 					: INT;						// type of the drive/cylinder/... that is to be operated by the valve ->  see list of drive types at support portal (www.festo.com/sp/)
	 	iDriveStroke 				: INT; 						// stroke of the drive/cylinder/... that is to be operated by the valve [1 digit = 1 mm for linear drives, 1 digit = 1° for rotary drives]
		iInstallationPositionDrive 	: INT;  	 				// inclination of the cylinder with reference to a horizontal installation position [1 digit = 0.01°, positive values = advancing upwards]
		iInPortRetracted_optional	: INT;						// Sensor port for detection of end position at pressurisation of outlet port 2 (retracted), value is number of the slot (beginning from 0 and including valve slots) * 10 + number of the port
		iInPortAdvanced_optional	: INT;						// Sensor port for detection of end position at pressurisation of outlet port 4 (advanced), value is number of the slot (beginning from 0 and including valve slots) * 10 + number of the port
	
	// application parameters                               	
		iLoadRetracting 			: INT;						// mass that is to be moved by the drive when retracting ((2) pressurised) [1 digit = 0.01 kg]
	 	iLoadAdvancing 				: INT; 						// mass that is to be moved by the drive when advancing ((4) pressurised) [1 digit = 0.01 kg]
		iMomentOfInertiaRetracting	: INT;						// Moment of inertia during for swivel drives when retratcting ((2) pressirised) [1 digit = 1 kg cm³]
		iMomentOfInertiaAdvancing	: INT;						// Moment of inertia during for swivel drives when advancing ((4) pressirised) [1 digit = 1 kg cm³]
		iSoftStartFunction			: INT := 1;					// flag to enable or disable the iSoftStartFunction; 0 = disabled, 1 = enabled

	//tuning parameters
		iOptProportionalGainFor2	: INT;						// Optional tuning parameter for the customized proportional element of the PID modulator at outlet port 2 [1 digit = 1 %]
		iOptProportionalGainFor4	: INT;						// Optional tuning parameter for the customized proportional element of the PID modulator at outlet port 4 [1 digit = 1 %]
		
	// function block response
		iResponse 					: eTransferResponse; 		// returns the status of the upload process
		xBusy						: BOOL;						// TRUE as long as the upload process is running
		xDone 						: BOOL; 					// indicates whether the upload was successfull
		xError 						: BOOL; 					// indicates whether an error occurred during the transfer
		xAborted					: BOOL;						// TRUE if the function block was canceled by xAbort	
END_VAR

VAR
	iState							: INT := 10;
	xStateChange					: BOOL;
	iCommandNumber					: INT;
	xFirstCycle						: BOOL := TRUE;				// indicator for the first cycle of the function block
	iParameterSetFC					: INT;						// value on input iParameterSet during first cycle
	
	aTransferPackages				: ARRAY [0..100] OF stTransferPackage;
	fbreadbitsfromword				: FB_Read_Bits_From_Word;
	fbuploadMultipleParameters 		: FB_Upload_Multiple_Parameters;
	fbWriteValueToWord 				: FB_Write_Value_To_Word;

	iCounterResetArray				: INT;

	iCurrentValveMode				: INT;						//
END_VAR

(*****************************************************************************************************

Festo SE & Co. KG, Esslingen
Copyright (c) 2021. All rights reserved.

Product:            Motion Terminal VTEM
Description:        Function Block to upload the parameters for Motion App 8 from the Motion Terminal

Object version:     2.00
Last change:        2021-07
======================================================================================================
                                       H I S T O R Y
======================================================================================================
Version:            2.00
Date:               2021-07
Change/Activity:    - created (#3872357)
Release:            3.5.7.237 (CODESYS 3.5.7.2, Lib version 3.7)
Author:             JEBU
======================================================================================================

*****************************************************************************************************)

// pre-check of the value for the parameter set
	IF xExecute = TRUE AND (iParameterSet < 1 OR iParameterSet > 5) THEN		// invalid input for the parameter set
		xDone := FALSE; 
		xError := TRUE; 
		iResponse := eTransferResponse.invalid_ParameterSet;
		xStateChange := TRUE;
		iState := 70;	// ERROR
	END_IF
//-----------------------------------------------------------------------------------------------------------

// check if iParameterSet was changed
	IF xExecute = TRUE AND xFirstCycle = TRUE THEN
		xFirstCycle := FALSE;
		iParameterSetFC := iParameterSet;
	END_IF
	
	IF xExecute = TRUE AND iParameterSet <> iParameterSetFC THEN
		xStateChange := TRUE;
		iState := 70;
		iResponse := eTransferResponse.FB_needs_rising_edge_xExecute;
	END_IF
//-----------------------------------------------------------------------------------------------------------

// WRITE PARAMETER INDICES INTO ARRAY
	//iTubingLengthAt2
		aTransferPackages[0].iChannel := iParameterSet;
		aTransferPackages[0].iAddressedTarget := 8;
		aTransferPackages[0].iIndex := 12;
		
	//iTubingLengthAt4
		aTransferPackages[1].iChannel := iParameterSet;
		aTransferPackages[1].iAddressedTarget := 8;
		aTransferPackages[1].iIndex := 13;
		
	//iTubingInnerDiameterAt2
		aTransferPackages[2].iChannel := iParameterSet;
		aTransferPackages[2].iAddressedTarget := 8;
		aTransferPackages[2].iIndex := 14;
		
	//iTubingInnerDiameterAt4
		aTransferPackages[3].iChannel := iParameterSet;
		aTransferPackages[3].iAddressedTarget := 8;
		aTransferPackages[3].iIndex := 15;
		
	//iDriveType
		aTransferPackages[4].iChannel := iParameterSet;
		aTransferPackages[4].iAddressedTarget := 8;
		aTransferPackages[4].iIndex := 20;
		
	//iDriveStroke
		aTransferPackages[5].iChannel := iParameterSet;
		aTransferPackages[5].iAddressedTarget := 8;
		aTransferPackages[5].iIndex := 21;
		
	//iInstallationPositionDrive
		aTransferPackages[6].iChannel := iParameterSet;
		aTransferPackages[6].iAddressedTarget := 8;
		aTransferPackages[6].iIndex := 60;
		
	//iLoadRetracting
		aTransferPackages[7].iChannel := iParameterSet;
		aTransferPackages[7].iAddressedTarget := 8;
		aTransferPackages[7].iIndex := 100;
		
	//iLoadAdvancing
		aTransferPackages[8].iChannel := iParameterSet;
		aTransferPackages[8].iAddressedTarget := 8;
		aTransferPackages[8].iIndex := 101;
		
	//iMomentOfInertiaRetracting
		aTransferPackages[9].iChannel := iParameterSet;
		aTransferPackages[9].iAddressedTarget := 8;
		aTransferPackages[9].iIndex := 102;
		
	//iMomentOfInertiaAdvancing
		aTransferPackages[10].iChannel := iParameterSet;
		aTransferPackages[10].iAddressedTarget := 8;
		aTransferPackages[10].iIndex := 103;
		
	//iSoftStartFunction
		aTransferPackages[11].iChannel := iParameterSet;
		aTransferPackages[11].iAddressedTarget := 8;
		aTransferPackages[11].iIndex := 222;
		
	//iInPortRetract_optional
		aTransferPackages[12].iChannel := iParameterSet;
		aTransferPackages[12].iAddressedTarget := 8;
		aTransferPackages[12].iIndex := 70;
		
	//iInPortAdvanced_optional
		aTransferPackages[13].iChannel := iParameterSet;
		aTransferPackages[13].iAddressedTarget := 8;
		aTransferPackages[13].iIndex := 71;
		
	//iOptProportionalGainFor2
		aTransferPackages[14].iChannel := iParameterSet;
		aTransferPackages[14].iAddressedTarget := 8;
		aTransferPackages[14].iIndex := 239;
		
